{region "Documentation"}
(*
Функциональный блок обработки аварии
====================================
:Date: 2019-11-21
Служит для отображения аварий в текущем списке аварий и ведения истории.
В одном проекте может быть обьявлено максимум 1000 функциональных блоков FB_Alarm.
Максимальная глубина журнала аварий 1000.

Принцип использования
=====================
1. В библиотеке есть готовые экземпляры визуализации с таблицей текущих активных аварий: *Current_Alarms*
	и журналом аварий *History_Alarms*. Их следует добавить в проект, если есть необходимость в графическом отображении.
2. Перед обьявлением экземпляров обязательно следует добавить в исполняемый код программу *PRG_Alarms_Core();* 	 
	В этой подпрограмме происходят вызовы всех экземпляров FB_Alarm, а также всё необходимое для корректной работы системы вцелом.
3. После объявления *FB_Alarm*. Все что требуется для его использования это задать параметры и аварийное условие.

4. По переднему фронту *fbAlarm.AlarmEvent* активируется аварийная блокировка ("1" на выходе fbAlarm.isActive).
	 По заднему фронту входа *fbAlarm.AlarmEvent*Аварийная блокировкка снимется ("0" на выходе fbAlarm.isActive) в зависимости от типа аварии: 
====================  ========================================================
Alarm_Type           	Поведение по заднему фронту *fbAlarm.AlarmEvent*
====================  ========================================================
Local_Quit       		Снимается только после локального квитирования аварии
	 					LibAlarms.bLocalQuitAllAlarms - глобальная переменная 
						сброса квитирования всех активных аварий
						fbAlarm.bQuitAlarm - квитирование аварии экземпляра ФБ                 		
Alarm_ScadaQuit    		Снимается только после локального квитирования аварии
	 					LibAlarms.bLocalQuitAllAlarms - глобальная переменная 
						сброса квитирования всех активных аварий
	 					LibAlarms.bRemoteQuitAllAlarms - глобальная переменная 
						сброса квитирования всех активных аварий 							 
						fbAlarm.bQuitAlarm - квитирование аварии экземпляра ФБ
Alarm_NoQuit	    	Снимается сразу по заднему фронту *fbAlarm.AlarmEvent*
	 					Если не была квитирована, то об этом появиться запись в
						журнале
Warning_RecordOnly   	Делает запись в журнал по переднему фронту *fbAlarm.AlarmEvent*
    	 			 	Снимается без квитирования.
===================   ========================================================
5. Для отображения списка текущих аварий нужно использовать диалоговое окно TcSakhnenko.Current_Allarms_dialog
	 Для отображения журнала аварий нужно использовать диалоговое окно TcSakhnenko.History_Of_Allarms_dialog
*)
{endregion}
FUNCTION_BLOCK FINAL FB_Alarm	
VAR_INPUT
	AlarmCheckIsEnable: 		BOOL:=TRUE;		(*Проверка аварийного условия активна*)
	AlarmEvent: 				BOOL:=FALSE; 	(*Условие срабатывания аварии*)
	bQuitAlarm:    				BOOL:=FALSE;	(*Команда на квитирование аварии, 1-квитирование*)
	AlarmType: 					AlarmType; 		(*Тип квитирования аварии*)
	AlarmInfo: ST_AlarmInfo; 
	AlarmActivationDelay: 		TIME; 			(*Задержка на срабатывание аварии*)
END_VAR
VAR_OUTPUT
	isActive: BOOL; 		(*Аварийая блокировка активна*)
	WasQuited: BOOL;		(*Авария была квитирована*)
END_VAR
VAR
	tDelay : TON;
	TempAlarmRec: ST_AlarmRecord;
	AlarmNum: UINT; 			(*Порядковый номер аварии*)
	iState: UINT;(*Состояние аварии*)
	i: UINT;
	n: UINT;
END_VAR

IF AlarmCheckIsEnable THEN 
	CASE  AlarmType OF
		00:
			a1_Local_Quit();
		01:
			a2_Alarm_ScadaQuit();
		02:
			a3_Alarm_NoQuit();
		03:
			a4_Warning_RecordOnly();
	END_CASE
END_IF

ACTION a1_Local_Quit:
(*Обработчик Аварии, которую необходимо квитировать. Только локально.*)
TempAlarmRec.wasQuited:=WasQuited;
TempAlarmRec.isActive:=isActive;

CASE iState OF
	0:(*Инициализация*)
		isActive:=FALSE;
		WasQuited:=FALSE;
		TempAlarmRec.wasQuited:=FALSE;
		TempAlarmRec.Time_Quit:="Не квитирована";
		TempAlarmRec.AlarmID:=AlarmInfo.AlarmID;
		TempAlarmRec.Color:=AlarmInfo.Color;
		TempAlarmRec.Description:=AlarmInfo.Description;
		TempAlarmRec.PossibleCause:=AlarmInfo.PossibleCause;
 		iState:=10;

	10:(*Авария не активна. Ожидание активации аварии*)
		tDelay(IN:=AlarmEvent, PT:=AlarmActivationDelay);
			
		IF tDelay.Q THEN (*Возникновение первой аварии*)
			TempAlarmRec.PossibleCause:=AlarmInfo.PossibleCause;
			tDelay(IN:=FALSE);
			iState:=20;
		END_IF

		IF isActive THEN (*Авария не была квитирована и возникла еще раз*)
			TempAlarmRec.PossibleCause:=AlarmInfo.PossibleCause;
			tDelay(IN:=FALSE);
			iState:=30;
		END_IF
		
	20: (*Запись Времени Аварии*)
		TempAlarmRec.Time_On:=LibAlarm.Global_TimeStr;
		isActive:=TRUE;
		iState:= 30;
		
	30: (*Ожидание квитирования аварии и ее ухода*)
		IF (LibAlarm.bLocalQuitAllAlarms OR bQuitAlarm) THEN 
			TempAlarmRec.Time_Quit:=LibAlarm.Global_TimeStr;
			WasQuited:=TRUE;
			iState:=40;
		END_IF

		IF NOT AlarmEvent THEN
			IF NOT WasQuited THEN
				TempAlarmRec.Time_OFF:=LibAlarm.Global_TimeStr;
				iState:=31;
			END_IF;
		END_IF
	31:(*Авария ушла но не квитирована*)
			IF (LibAlarm.bLocalQuitAllAlarms OR bQuitAlarm) THEN
				TempAlarmRec.Time_Quit:=LibAlarm.Global_TimeStr;
				WasQuited:=TRUE;

				FOR i:=0 TO (LibAlarm.MAX_HISTORY_NUM - 2) DO
					n:=LibAlarm.MAX_HISTORY_NUM-i;
					LibAlarm.HistoryAlarmsArray[n]:=LibAlarm.HistoryAlarmsArray[n-1];
				END_FOR;

				LibAlarm.HistoryAlarmsArray[1]:=TempAlarmRec;
				iState:=00;
			END_IF
		
		IF AlarmEvent THEN //авария пришла снова
			TempAlarmRec.Time_Quit:="Не квитирована";

			FOR i:=0 TO (LibAlarm.MAX_HISTORY_NUM - 2) DO
				n:=LibAlarm.MAX_HISTORY_NUM-i;
				LibAlarm.HistoryAlarmsArray[n]:=LibAlarm.HistoryAlarmsArray[n-1];
			END_FOR;
		
			LibAlarm.HistoryAlarmsArray[1]:=TempAlarmRec;
			
			iState:=10;
		END_IF
		
		40:(*Авария ушла и квитирована*)
			IF NOT AlarmEvent THEN
			TempAlarmRec.Time_OFF:=LibAlarm.Global_TimeStr;

				FOR i:=0 TO (LibAlarm.MAX_HISTORY_NUM - 2) DO
					n:=LibAlarm.MAX_HISTORY_NUM-i;
					LibAlarm.HistoryAlarmsArray[n]:=LibAlarm.HistoryAlarmsArray[n-1];
				END_FOR;
		
				LibAlarm.HistoryAlarmsArray[1]:=TempAlarmRec;

				iState:=0;
			END_IF
		
END_CASE
END_ACTION

ACTION a2_Alarm_ScadaQuit:
(*Обработчик Аварии, которую необходимо квитировать. Локально и удаленно.*)
TempAlarmRec.wasQuited:=WasQuited;
TempAlarmRec.isActive:=isActive;

CASE iState OF
	0:(*Инициализация*)
		isActive:=FALSE;
		WasQuited:=FALSE;
		TempAlarmRec.Time_Quit:="Не квитирована";
		TempAlarmRec.AlarmID:=AlarmInfo.AlarmID;
		TempAlarmRec.Color:=AlarmInfo.Color;
		TempAlarmRec.Description:=AlarmInfo.Description;
		TempAlarmRec.PossibleCause:=AlarmInfo.PossibleCause;
 		iState:=10;

	10:(*Авария не активна. Ожидание активации аварии*)
		tDelay(IN:=AlarmEvent, PT:=AlarmActivationDelay);
			
		IF tDelay.Q THEN (*Возникновение первой аварии*)
			TempAlarmRec.PossibleCause:=AlarmInfo.PossibleCause;
			tDelay(IN:=FALSE);
			iState:=20;
		END_IF

		IF isActive THEN (*Авария не была квитирована и возникла еще раз*)
			TempAlarmRec.PossibleCause:=AlarmInfo.PossibleCause;
			tDelay(IN:=FALSE);
			iState:=30;
		END_IF
		
	20: (*Запись Времени Аварии*)
		TempAlarmRec.Time_On:=LibAlarm.Global_TimeStr;
		isActive:=TRUE;
		iState:= 30;
		
	30: (*Ожидание квитирования аварии и ее ухода*)
		IF (LibAlarm.bLocalQuitAllAlarms OR bQuitAlarm OR LibAlarm.bRemoteQuitAllAlarms) THEN 
			TempAlarmRec.Time_Quit:=LibAlarm.Global_TimeStr;
			WasQuited:=TRUE;
			iState:=40;
		END_IF

		IF NOT AlarmEvent THEN
			IF NOT WasQuited THEN
				TempAlarmRec.Time_OFF:=LibAlarm.Global_TimeStr;
				iState:=31;
			END_IF;
		END_IF
	31:(*Авария ушла но не квитирована*)
			IF (LibAlarm.bLocalQuitAllAlarms OR bQuitAlarm OR LibAlarm.bRemoteQuitAllAlarms) THEN
				TempAlarmRec.Time_Quit:=LibAlarm.Global_TimeStr;
				WasQuited:=TRUE;

				FOR i:=0 TO (LibAlarm.MAX_HISTORY_NUM - 2) DO
					n:=LibAlarm.MAX_HISTORY_NUM-i;
					LibAlarm.HistoryAlarmsArray[n]:=LibAlarm.HistoryAlarmsArray[n-1];
				END_FOR;

				LibAlarm.HistoryAlarmsArray[1]:=TempAlarmRec;
				iState:=00;
			END_IF

		IF AlarmEvent THEN
			TempAlarmRec.Time_Quit:="Не квитирована";

			FOR i:=0 TO (LibAlarm.MAX_HISTORY_NUM - 2) DO
				n:=LibAlarm.MAX_HISTORY_NUM-i;
				LibAlarm.HistoryAlarmsArray[n]:=LibAlarm.HistoryAlarmsArray[n-1];
			END_FOR;
		
			LibAlarm.HistoryAlarmsArray[1]:=TempAlarmRec;
			
			iState:=10;
		END_IF
		
		40:(*Авария ушла и квитирована*)
			IF NOT AlarmEvent THEN
			TempAlarmRec.Time_OFF:=LibAlarm.Global_TimeStr;

				FOR i:=0 TO (LibAlarm.MAX_HISTORY_NUM - 2) DO
					n:=LibAlarm.MAX_HISTORY_NUM-i;
					LibAlarm.HistoryAlarmsArray[n]:=LibAlarm.HistoryAlarmsArray[n-1];
				END_FOR;
		
				LibAlarm.HistoryAlarmsArray[1]:=TempAlarmRec;

				iState:=0;
			END_IF
		
END_CASE
END_ACTION

ACTION a3_Alarm_NoQuit:
(*Обработчик Аварии, которую необходимо квитировать*)
TempAlarmRec.wasQuited:=WasQuited;
TempAlarmRec.isActive:=isActive;

CASE iState OF
	0:(*Инициализация*)
		isActive:=FALSE;
		WasQuited:=FALSE;
		TempAlarmRec.Time_Quit:="Не квитирована";
		TempAlarmRec.AlarmID:=AlarmInfo.AlarmID;
		TempAlarmRec.Color:=AlarmInfo.Color;
		TempAlarmRec.Description:=AlarmInfo.Description;
		TempAlarmRec.PossibleCause:=AlarmInfo.PossibleCause;
 		iState:=10;

	10:(*Авария не активна. Ожидание активации аварии*)
		tDelay(IN:=AlarmEvent, PT:=AlarmActivationDelay);
			
		IF tDelay.Q THEN (*Возникновение первой аварии*)
			TempAlarmRec.PossibleCause:=AlarmInfo.PossibleCause;
			tDelay(IN:=FALSE);
			iState:=20;
		END_IF

		IF isActive THEN (*Авария не была квитирована и возникла еще раз*)
			TempAlarmRec.PossibleCause:=AlarmInfo.PossibleCause;
			tDelay(IN:=FALSE);
			iState:=30;
		END_IF
		
	20: (*Запись Времени Аварии*)
		TempAlarmRec.Time_On:=LibAlarm.Global_TimeStr;
		isActive:=TRUE;
		iState:= 30;
		
	30: (*Ожидание квитирования аварии и ее ухода*)
		IF (LibAlarm.bLocalQuitAllAlarms OR bQuitAlarm OR LibAlarm.bRemoteQuitAllAlarms) THEN 
			TempAlarmRec.Time_Quit:=LibAlarm.Global_TimeStr;
			WasQuited:=TRUE;
			iState:=40;
		END_IF

		IF NOT AlarmEvent THEN
			IF NOT WasQuited THEN
				TempAlarmRec.Time_OFF:=LibAlarm.Global_TimeStr;
				iState:=40;
			END_IF;
		END_IF
		
		40:(*Авария ушла и квитирована*)
			IF NOT AlarmEvent THEN
			TempAlarmRec.Time_OFF:=LibAlarm.Global_TimeStr;

				FOR i:=0 TO (LibAlarm.MAX_HISTORY_NUM - 2) DO
					n:=LibAlarm.MAX_HISTORY_NUM-i;
					LibAlarm.HistoryAlarmsArray[n]:=LibAlarm.HistoryAlarmsArray[n-1];
				END_FOR;
		
				LibAlarm.HistoryAlarmsArray[1]:=TempAlarmRec;

				iState:=0;
			END_IF
		
END_CASE
END_ACTION

ACTION a4_Warning_RecordOnly:
(*Предупреждение*)
CASE iState OF
	0:(*Инициализация*)
		isActive:=FALSE;
		WasQuited:=FALSE;
		TempAlarmRec.Time_Quit:="Не квитирована";
		TempAlarmRec.AlarmID:=AlarmInfo.AlarmID;
		TempAlarmRec.Color:=AlarmInfo.Color;
		TempAlarmRec.Description:=AlarmInfo.Description;
		TempAlarmRec.PossibleCause:=AlarmInfo.PossibleCause;
 		iState:=10;

	10:(*Авария не активна. Ожидание активации аварии*)
		tDelay(IN:=AlarmEvent, PT:=AlarmActivationDelay);
			
		IF tDelay.Q THEN (*Возникновение первой аварии*)
			tDelay(IN:=FALSE);
			
			TempAlarmRec.Time_ON:=LibAlarm.Global_TimeStr;
			TempAlarmRec.Time_Quit:="Не квитирована";
			TempAlarmRec.Time_OFF:=LibAlarm.Global_TimeStr;
			
				FOR i:=0 TO (LibAlarm.MAX_HISTORY_NUM - 2) DO
					n:=LibAlarm.MAX_HISTORY_NUM-i;
					LibAlarm.HistoryAlarmsArray[n]:=LibAlarm.HistoryAlarmsArray[n-1];
				END_FOR;
		
				LibAlarm.HistoryAlarmsArray[1]:=TempAlarmRec;
				
			iState:=20;
		END_IF

		
	20: (*Запись Времени Аварии*)
		IF NOT AlarmEvent THEN
			iState:=00;
		END_IF
		
END_CASE
END_ACTION

METHOD FB_init : BOOL
VAR_INPUT
	bInitRetains : BOOL; // if TRUE, the retain variables are initialized (warm start / cold start)
	bInCopyCode : BOOL;  // if TRUE, the instance afterwards gets moved into the copy code (online change)
END_VAR
libAlarm.iNumberOfAlarms:=libAlarm.iNumberOfAlarms+1;
AlarmNum:=libAlarm.iNumberOfAlarms;
LibAlarm.FB_Alarm_Iterator[AlarmNum]:=THIS;
END_METHOD

END_FUNCTION_BLOCK

(* stored: Version 1.1.0.1, ProductVersion 3.1.4024.9
   POU FB_Alarm: Id {969aa0c0-5b48-4116-b2b9-42f210740f10}, SpecialFunc None
   Action a1_Local_Quit: Id {63db822d-757d-41d1-a186-386720b24979}
   Action a2_Alarm_ScadaQuit: Id {b1187035-1c17-4f98-b40e-69d35d0a67ff}
   Action a3_Alarm_NoQuit: Id {9e00bcd7-b8a4-429b-b0aa-2b69a42f477c}
   Action a4_Warning_RecordOnly: Id {c1e311af-8afc-43bc-8c63-a7e2e0019169}
   Method FB_init: Id {85054220-a632-4910-bba1-a4c748b42899} *)
